TYPE ST_TCPConnection_IO :
STRUCT
END_STRUCT
END_TYPE

(* stored: Version 1.1.0.1, ProductVersion 3.1.4024.12
   DUT ST_TCPConnection_IO: Id {339247d8-95a1-4670-be8f-1322ec643be3} *)
